{attribute 'qualified_only'}
VAR_GLOBAL
	vari : int;
END_VAR

(* stored: Version 1.1.0.1, ProductVersion 3.1.4024.9
   GVL GVL: Id {885db123-f76c-438c-a428-6f198b1b2929} *)
